{attribute 'linkalways'} 
{attribute 'no_explicit_call' := 'This FB is a CLASS and must be accessed using methods or properties'}
{attribute 'enable_dynamic_creation'}
FUNCTION_BLOCK _USINT EXTENDS DatatypeBase
VAR
	localData : USINT;
	activeData : REFERENCE TO USINT REF= localData;
END_VAR

PROPERTY PUBLIC Address : PVOID
GET
Address := ADR(activeData);
END_GET
END_PROPERTY

METHOD PUBLIC ClearReference
VAR_INPUT
END_VAR
activeData REF= localData;
END_METHOD

METHOD PUBLIC Clone : I_Datatype
VAR
    pClone : POINTER TO _USINT;
END_VAR
pClone := __NEW(_USINT(InitialValue := Value));
Clone := pClone^;
END_METHOD

METHOD FB_init : BOOL
VAR_INPUT
	bInitRetains : BOOL; // if TRUE, the retain variables are initialized (warm start / cold start)
	bInCopyCode : BOOL;  // if TRUE, the instance afterwards gets moved into the copy code (online change)
	InitialValue : USINT;
END_VAR
localData := InitialValue;
END_METHOD

PROPERTY PUBLIC IecType : T_MAXSTRING
GET
IecType := 'USINT';
END_GET
END_PROPERTY

METHOD PUBLIC MakeReferenceTo
VAR_INPUT
	ReferenceTarget : REFERENCE TO USINT;
END_VAR
activeData REF= ReferenceTarget;
END_METHOD

METHOD PUBLIC SerializeWith
VAR_INPUT
	Serializer : I_Serializer;
END_VAR
Serializer.AddUsint(activeData);
END_METHOD

PROPERTY PUBLIC Size : UDINT
GET
Size := SIZEOF(activeData);
END_GET
END_PROPERTY

METHOD TryDeserializeFrom : BOOL
VAR_INPUT
	Deserializer : I_Deserializer;
	Feedback : I_DeserializerFeedback;
END_VAR
TryDeserializeFrom := Deserializer.TryGetUsint(activeData, Feedback);
END_METHOD

METHOD TryMakeReferenceTo : BOOL
VAR_INPUT
	Target : I_Datatype;
END_VAR
VAR
	pTargetData : POINTER TO USINT;
END_VAR
IF NOT (Target.IecType = IecType) THEN
	RETURN;
END_IF

pTargetData := Target.Address;
activeData REF= pTargetData^;
TryMakeReferenceTo := TRUE;
END_METHOD

PROPERTY PUBLIC Value : USINT
GET
Value := activeData;
END_GET
SET
activeData := Value;
END_SET
END_PROPERTY

END_FUNCTION_BLOCK

(* stored: Version 1.1.0.1, ProductVersion 3.1.4024.12
   POU _USINT: Id {73d9601c-574b-01d1-23fa-d23608a3f39d}, SpecialFunc None
   Folder Constructor: Id {8ea448e0-ef12-02b0-09a6-a0d856d04e10}
   Property Address: Id {c6c4df9a-ed9d-0878-0493-207e41e8a267}
   Get Get: Id {aed9dd39-95b9-0a36-0d45-aa6e7e12e1fd}
   Method ClearReference: Id {21ba2945-92c3-019d-043a-7783a1082725}
   Method Clone: Id {df97922d-f0b2-02bf-2307-02d5de55f866}
   Method FB_init: Id {d6617acf-b88a-0d8d-1863-8dfae5b8e461}
   Property IecType: Id {e4dae87d-f3e5-0db5-2664-254a92afcf0a}
   Get Get: Id {4db4257f-630e-088b-31d7-2c9341d8f5b9}
   Method MakeReferenceTo: Id {7160aee3-8c59-0f96-1d92-b5d6ffc1710e}
   Method SerializeWith: Id {fa2ec0ce-951b-0bad-147a-00375cea3f94}
   Property Size: Id {d8011a71-b0ed-0106-3a73-7aad696a0038}
   Get Get: Id {6e611b70-7153-03fa-24c8-1a6fa7f9ecab}
   Method TryDeserializeFrom: Id {9491981d-c6cd-07bd-0538-6e067b4c6752}
   Method TryMakeReferenceTo: Id {8b0b5ccc-8127-02e6-025f-dccf2058d158}
   Property Value: Id {c58e94f1-6676-00ff-043e-8bb7a8e13261}
   Get Get: Id {1d887d9e-eb5a-0289-0fc4-9e5c5b1c4ca7}
   Set Set: Id {b25991f3-88b1-0f6e-2f45-128fb27b28f1} *)
